{attribute 'GeneratedUsingTerminal: EK1100-0000-0018'}
{attribute addProperty BoxType "EK1100-0000-0018"}
{attribute addProperty Id "Beckhoff_EPP6xxxEK1122Beckhoff_EPP6xxxEK1122_484AACC3672"}
{attribute addProperty CRC "1246990091"}
{attribute addProperty Size "672"}
TYPE Beckhoff_EPP6xxx_4A538F0B EXTENDS EK1100_1FC0878B :
STRUCT
	{attribute addProperty Name "Beckhoff_EPP6xxxEK1122"}
	{attribute addProperty PreviousPort "Beckhoff EPP6xxx : B"}
	Beckhoff_EPP6xxxEK1122 : Beckhoff_EPP6xxxEK1122_484AACC3;
END_STRUCT
END_TYPE

(* stored: Version 1.2.0.0, ProductVersion 3.1.4024.9
   DUT Beckhoff_EPP6xxx_4A538F0B: Id {ffd4429a-d16c-4d2c-a5e0-886dbbfb2bf5} *)
